{attribute 'GeneratedUsingTerminal: EK1122-0000-0018'}
{attribute addProperty BoxType "EK1122-0000-0018"}
{attribute addProperty Id "Beckhoff_EJ3xxxsub_EK1100EK1100_AB5A94672"}
{attribute addProperty CRC "4100403987"}
{attribute addProperty Size "2"}
TYPE Beckhoff_EJ3xxxEK1122_F4673313 EXTENDS EK1122_AB5A9467 :
STRUCT
	{attribute addProperty Name "Beckhoff_EJ3xxxsub_EK1100"}
	Beckhoff_EJ3xxxsub_EK1100 : EK1100_AB5A9467;
END_STRUCT
END_TYPE

(* stored: Version 1.2.0.0, ProductVersion 3.1.4024.9
   DUT Beckhoff_EJ3xxxEK1122_F4673313: Id {3426db10-0498-4643-b0b3-03af86102be8} *)
